PROGRAM TestRunner
VAR
	test_wrapper : TestWrapper;
	date_time_time : DateTime_Test;
	helper_functions_test : ConvertAnyToString_Test;
	dynamic_string_buffer_test : DynamicStringBuffer_Test;
END_VAR

test_wrapper();

TcUnit.Run();

END_PROGRAM

(* stored: Version 1.1.0.1, ProductVersion 3.1.4026.17
   POU TestRunner: Id {379526ca-9719-4af5-b69e-537f4c5508c9}, SpecialFunc None *)
